PROGRAM MAIN
VAR
END_VAR

END_PROGRAM

(* stored: Version 1.1.0.1
   POU MAIN: Id {f3413dde-4def-4abb-bcf5-29bbf0cae88d} *)
